TYPE GroupBoxLayout:
STRUCT
	{attribute wpf [Container(Layout.Stack)]}
	{attribute wpf [Group(Layout.GroupBox)]}
	{attribute addProperty Name "<#Various types#>"}
	_vt: VariousTypes;
END_STRUCT
END_TYPE

(* stored: Version 1.1.0.1, ProductVersion 3.1.4024.9
   DUT GroupBoxLayout: Id {cad173a1-4b25-44ff-9267-9295204f781a} *)
